SUBAPPLICATION Uebung_012b (* Numeric Value Input und Speichern *)
  (* Standard: 61499-2; Description: Copyright (c) 2023 Meisterschulen am Ostbahnhof This program and the accompanying materials are made available under the terms of the Eclipse Public License 2.0 which is available at https://www.eclipse.org/legal/epl-2.0/ SPDX-License-Identifier: EPL-2.0 *)
  (* Version 1.0, 2023-10-23, Franz Höpfinger, Meisterschulen am Ostbahnhof *)
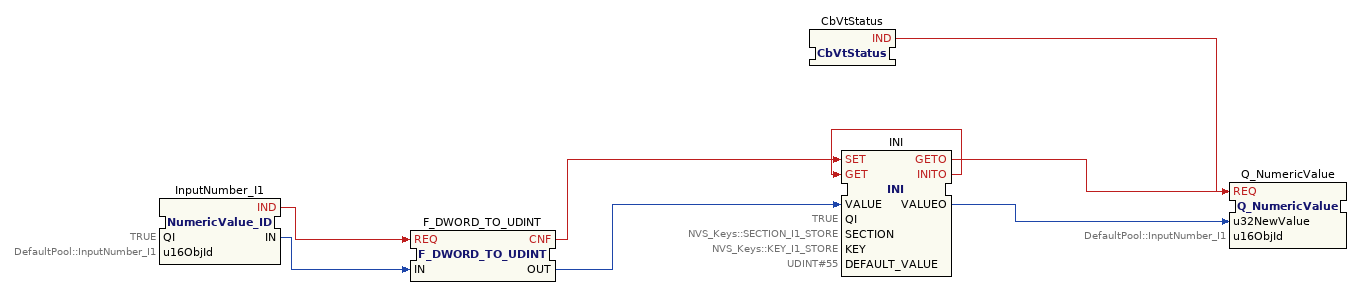
  FBS
    F_DWORD_TO_UDINT : F_DWORD_TO_UDINT;
    InputNumber_I1 : NumericValue_ID(QI := TRUE, u16ObjId := DefaultPool::InputNumber_I1);
    INI : INI(QI := TRUE, SECTION := NVS_Keys::SECTION_I1_STORE, KEY := NVS_Keys::KEY_I1_STORE, DEFAULT_VALUE := UDINT#55);
    Q_NumericValue : Q_NumericValue(u16ObjId := DefaultPool::InputNumber_I1);
    CbVtStatus : CbVtStatus;
  END_FBS
  EVENT_CONNECTIONS
    InputNumber_I1.IND TO F_DWORD_TO_UDINT.REQ;
    F_DWORD_TO_UDINT.CNF TO INI.SET;
    INI.GETO TO Q_NumericValue.REQ;
    CbVtStatus.IND TO Q_NumericValue.REQ;
    INI.INITO TO INI.GET;
  END_CONNECTIONS
  DATA_CONNECTIONS
    InputNumber_I1.IN TO F_DWORD_TO_UDINT.IN;
    F_DWORD_TO_UDINT.OUT TO INI.VALUE;
    INI.VALUEO TO Q_NumericValue.u32NewValue;
  END_CONNECTIONS
END_SUBAPPLICATION
